TYPE "Positioning_EPOS_Machine_Wng"
VERSION : 0.1
// Block: Positioning_EPOS_Machine_Wng
   STRUCT
      NotAutReady : Bool;
      Minus_CndMissing : Bool;
      Plus_CndMissing : Bool;
      S120_Warning : Bool;
      Ax_NotHomed : Bool;
      Ax_FlyingHome : Bool;
      Ax_SwLimitMinus : Bool;
      Ax_SwLimitPlus : Bool;
   END_STRUCT;

END_TYPE
